// TIA Portal V21 export
// export: Created 2026-07-07T09:15:55.8352405Z, ExportSetting WithReadOnly, DisplayName Totally Integrated Automation Portal, DisplayVersion V21, DisplayName SINAMICS Startdrive Advanced, DisplayVersion V21, DisplayName SINAMICS Startdrive G110M, G120, G120C, G120D, G120P, G115D, DisplayVersion V21, DisplayName SINAMICS Startdrive G130, G150, S120, S150, G200, G220, S200, S210, S220, Innomotics MVD, DisplayVersion V21, DisplayName STEP 7 Professional, DisplayVersion V21, DisplayName STEP 7 Safety, DisplayVersion V21, DisplayName Tech WebApplication, DisplayVersion V21, DisplayName WinCC Basic/Comfort/Advanced, DisplayVersion V21, DisplayName WinCC Professional, DisplayVersion V21, DisplayName WinCC Unified, DisplayVersion V21
Screen "Screen_03_PID_Settings"  Nonex480, Template=模板_1
  ScreenLayer 
    TextField "Title" at 20,12 size 760x34  Text="画面 3：参数设置画面"
    TextField "NavBar" at 20,430 size 760x34  Text="主监控 手动调试 参数设置 报警诊断 趋势"
    TextField "Hdr_EC_PID_288" at 20,60 size 240x26  Text="EC PID"
    TextField "Body_EC_PID_304" at 20,84 size 240x126  Text="Kp_EC_Set | Ki_EC_Set | Kd_EC_Set | EC_Trim_Band | Active_EC_SP"
    TextField "Hdr_pH_PID_320" at 280,60 size 240x26  Text="pH PID"
    TextField "Body_pH_PID_336" at 280,84 size 240x126  Text="Kp_pH_Set | Ki_pH_Set | Kd_pH_Set | pH_Trim_Band | Active_pH_SP"
    TextField "Hdr_N_P_K_352" at 540,60 size 240x26  Text="N/P/K 配方"
    TextField "Body_N_P_K_368" at 540,84 size 240x126  Text="N_Enable / N_Ratio / N_Max | P_Enable / P_Ratio / P_Max | K_Enable / K_Ratio / K_Max"
    TextField "Hdr_Item_384" at 20,230 size 500x26  Text="阶段与策略"
    TextField "Body_Item_400" at 20,254 size 500x126  Text="Growth_Stage | Stage_Auto_SP_Enable | Stage_EC_SP | Stage_pH_SP | Setpoint_Protection_Active"
    TextField "Hdr_Item_416" at 540,230 size 240x26  Text="执行通道参考"
    TextField "Body_Item_432" at 540,254 size 240x126  Text="N_Target / N_Actual / q_n_cmd | P_Target / P_Actual / q_p_cmd | K_Target / K_Actual / q_k_cmd"
